(* IEC 61131-3 sources: CodesysTest/export/Unused/FB_SimBasicSealFlatteners.pou/InPosition.prop, 1 file *)

(* ---- Get.pm.st ---- *)
(*#-#-#-#-#-#-#-#-#-#---Declaration---#-#-#-#-#-#-#-#-#-#-#-#-#*)

VAR
END_VAR
(*#-#-#-#-#-#-#-#-#-#---Implementation---#-#-#-#-#-#-#-#-#-#-#-#-#*)

InPosition := 	moveToBagFeed.Q OR
				moveToBagHolding.Q OR
				moveToClearance.Q OR
				moveToSeal.Q OR
				moveToIn.Q;
